(* IEC 61131-3 sources: ics/BLR101_ProenixContact/BLR101_1_ILC171_44/LogicalPOUs/Valve, 2 files *)

(* ---- ValveFB.ST ---- *)
(*@PROPERTIES_EX@
TYPE: POU
LOCALE: 0
IEC_LANGUAGE: ST
PLC_TYPE: independent
PROC_TYPE: independent
GROUP: Valve
*)
(*@KEY@:DESCRIPTION*)

(*@KEY@:END_DESCRIPTION*)
FUNCTION_BLOCK ValveFB

(*Group:Default*)

VAR
    Fb_Alrm_Tmr :	TON;
END_VAR

VAR_IN_OUT
    Vlv_strct :	Vlv;
END_VAR

VAR
    AlrmNotMove :	BOOL;
    AlrmSQ :	BOOL;
    RunManual :	BOOL;
    RunAuto :	BOOL;
    COM_Open :	BOOL;
    COM_Close :	BOOL;
END_VAR

VAR_INPUT
    SetOvertime :	TIME;
    Cycle :	Cycle;
END_VAR

VAR
    NotMove_Alrm_Tmr :	TON;
    AlrmFeedBack :	BOOL;
    AlarmBlock :	BOOL;
END_VAR

(*@KEY@: WORKSHEET
NAME: ValveFB
IEC_LANGUAGE: ST
*)
    (*Alarm processing*)
Fb_Alrm_Tmr(IN:=Vlv_strct.CW.Enable and (COM_Close or COM_Open) and not
    Vlv_strct.SW.RUN, PT:=t#3s);

NotMove_Alrm_Tmr(IN:=Vlv_strct.CW.Enable and
    ((COM_Close and not Vlv_strct.SW.Closed) or
    (COM_Open and not Vlv_strct.SW.Opened)),PT:=SetOvertime);

if Fb_Alrm_Tmr.Q then
    AlrmFeedBack:=true;
end_if;

if NotMove_Alrm_Tmr.Q then
    AlrmNotMove:=true;
end_if;

if (not Vlv_strct.CW.ExtraEn and (Vlv_strct.SW.COM_Open or Vlv_strct.SW.COM_Close)) then
    AlarmBlock:= true;
end_if;

if Vlv_strct.SW.Opened and Vlv_strct.SW.Closed then
    AlrmSQ:=true;
end_if;

if AlrmNotMove or AlrmSQ or AlrmFeedBack or Vlv_strct.CW.ExtraAlarm then
    Vlv_strct.SW.AlarmAccum:=true;
end_if;

if Vlv_strct.CW.ACK then
    Vlv_strct.SW.AlarmAccum:=false;
    AlrmFeedBack:=false;
    AlrmSQ:=false;
    AlrmnotMove:=false;
    AlarmBlock:= false;
end_if;

    (*Auto/Manual mode selection*)
if Vlv_strct.CW.EnableAuto then
    Vlv_strct.SW.Auto:= true;
end_if;
if Vlv_strct.CW.DisableAuto then
    Vlv_strct.SW.Auto:= false;
end_if;

Vlv_strct.SW.ManOK:=not Vlv_strct.SW.AlarmAccum and Vlv_strct.CW.AuxON and
    Vlv_strct.CW.Enable and not Vlv_strct.SW.Auto;

Vlv_strct.SW.AutoOK:= not Vlv_strct.SW.AlarmAccum and Vlv_strct.CW.AuxON and
    Vlv_strct.CW.Enable and Vlv_strct.SW.Auto and Cycle.SW.Running;

    (*Manual mode activation*)
if Vlv_strct.CW.ManOpen or Vlv_strct.CW.ManClose then
    RunManual:=true;
end_if;

if Vlv_strct.CW.Stop or not Vlv_strct.SW.ManOK then
    RunManual:=false;
end_if;

    (*Auto mode activation*)
RunAuto:= (Cycle.CW.PulseStart or RunAuto) and Vlv_strct.SW.AutoOK and
    Vlv_strct.SW.Auto;

    (*Set command for start*)
COM_Open:=((Vlv_strct.CW.AutoOpen and RunAuto and Vlv_strct.SW.AutoOK) or
    ((Vlv_strct.CW.ManOpen or COM_Open) and RunManual and Vlv_strct.SW.ManOK)) and not
    COM_Close and not Vlv_strct.SW.Opened;

COM_Close:=((Vlv_strct.CW.AutoClose and RunAuto and Vlv_strct.SW.AutoOK) or
    ((Vlv_strct.CW.ManClose or COM_Close) and RunManual and Vlv_strct.SW.ManOK)) and not
    COM_Open and not Vlv_strct.SW.Closed;

Vlv_strct.SW.COM_Open:=COM_Open and not Vlv_strct.CW.SimEn;
Vlv_strct.SW.COM_Close:=COM_Close and not Vlv_strct.CW.SimEn;

    (*Status processing*)
if Vlv_strct.SW.AlarmAccum then
    Vlv_strct.Status:=word#4;
elsif not Vlv_strct.CW.ExtraEn then
    Vlv_strct.Status:=word#8;
elsif Vlv_strct.SW.Opened then
    Vlv_strct.Status:=word#1;
elsif Vlv_strct.SW.Closed then
    Vlv_strct.Status:=word#2;
else
    Vlv_strct.Status:=word#0;
end_if;

Vlv_strct.CW.EnableAuto:=false;
Vlv_strct.CW.DisableAuto:=false;
Vlv_strct.CW.ManOpen:=false;
Vlv_strct.CW.Stop:=false;
Vlv_strct.CW.ManClose:=false;
Vlv_strct.CW.ACK:=false;

(*@KEY@: END_WORKSHEET *)
END_FUNCTION_BLOCK

(* ---- Valve_section.ST ---- *)
(*@PROPERTIES_EX@
TYPE: POU
LOCALE: 0
IEC_LANGUAGE: ST
PLC_TYPE: independent
PROC_TYPE: independent
GROUP: Valve
*)
(*@KEY@:DESCRIPTION*)

(*@KEY@:END_DESCRIPTION*)
PROGRAM Valve_section

(*Group:Default*)

VAR
    Vlv_Blr_in :	ValveFB;
    Vlv_Blr_out :	ValveFB;
    Exhsr_Gate :	ValveFB;
END_VAR

VAR_EXTERNAL
    Boiler :	Blr;
    Cycle :	Cycle;
    xVlv_in_QM_ON :	BOOL;
    xVlv_in_Remote :	BOOL;
    xVlv_in_RUN :	BOOL;
    xVlv_in_TorqueSwAlrm :	BOOL;
    xVlv_in_Closed :	BOOL;
    xVlv_in_Opened :	BOOL;
    xVlv_out_QM_ON :	BOOL;
    xVlv_out_Remote :	BOOL;
    xVlv_out_RUN :	BOOL;
    xVlv_out_TorqueSwAlrm :	BOOL;
    xVlv_out_Closed :	BOOL;
    xVlv_out_Opened :	BOOL;
    xExhsrGt_QM_ON :	BOOL;
    xExhsrGt_Remote :	BOOL;
    xExhsrGt_RUN :	BOOL;
    xExhsrGt_Closed :	BOOL;
    xExhsrGt_Opened :	BOOL;
    xVlv_in_COM_OP :	BOOL;
    xVlv_in_COM_CL :	BOOL;
    xVlv_out_COM_OP :	BOOL;
    xVlv_out_COM_CL :	BOOL;
    xExhsrGt_COM_OP :	BOOL;
    xExhsrGt_COM_CL :	BOOL;
    arrMB_Srv1Data :	MB2_TCP_ARR_W_0_7167;
    ExhsrGatePos :	Snsr;
END_VAR

VAR
    ExhsrGatePID :	BACL_PID3P_T1_V0_10;
END_VAR

(*@KEY@: WORKSHEET
NAME: Valve_section
IEC_LANGUAGE: ST
*)

    (*Boiler Input Valve DI*)
Boiler.V[1].CW.Enable:= xVlv_in_Remote;
Boiler.V[1].CW.AuxON:= Cycle.CW.AuxON;
Boiler.V[1].CW.ExtraEn:= xVlv_in_QM_ON;
Boiler.V[1].CW.ExtraAlarm:= not xVlv_in_TorqueSwAlrm;
Boiler.V[1].SW.Rem:= xVlv_in_Remote;
Boiler.V[1].SW.RUN:= xVlv_in_RUN;
Boiler.V[1].SW.Closed:= xVlv_in_Closed;
Boiler.V[1].SW.Opened:= xVlv_in_Opened;

    (*Boiler Input Valve FB call*)
Vlv_Blr_in(Vlv_strct:=Boiler.V[1],SetOvertime:=t#80s,Cycle:=Cycle);
Boiler.V[1]:=Vlv_Blr_in.Vlv_strct;
    (*ModBusArray ControlWord Reset*)
arrMB_Srv1Data[1492]:=word#0;

    (*Boiler Input Valve D0*)
xVlv_in_COM_OP:= Boiler.V[1].SW.COM_Open;
xVlv_in_COM_CL:= Boiler.V[1].SW.COM_Close;

    (*Boiler Output Valve DI*)
Boiler.V[2].CW.Enable:= xVlv_out_Remote;
Boiler.V[2].CW.AuxON:= Cycle.CW.AuxON;
Boiler.V[2].CW.ExtraEn:= xVlv_out_QM_ON;
Boiler.V[2].CW.ExtraAlarm:= not xVlv_out_TorqueSwAlrm;
Boiler.V[2].SW.Rem:= xVlv_out_Remote;
Boiler.V[2].SW.RUN:= xVlv_out_RUN;
Boiler.V[2].SW.Closed:= xVlv_out_Closed;
Boiler.V[2].SW.Opened:= xVlv_out_Opened;

    (*Boiler Output Valve FB call*)
Vlv_Blr_out(Vlv_strct:=Boiler.V[2],SetOvertime:=t#80s,Cycle:=Cycle);
Boiler.V[2]:=Vlv_Blr_out.Vlv_strct;
    (*ModBusArray ControlWord Reset*)
arrMB_Srv1Data[1508]:=word#0;

    (*Boiler Output Valve D0*)
xVlv_out_COM_OP:= Boiler.V[2].SW.COM_Open;
xVlv_out_COM_CL:= Boiler.V[2].SW.COM_Close;

    (*Exhauser Gate DI*)
Boiler.V[3].CW.Enable:= xExhsrGt_Remote;
Boiler.V[3].CW.AuxON:= Cycle.CW.AuxON;
Boiler.V[3].CW.ExtraEn:= xExhsrGt_QM_ON;
Boiler.V[3].SW.Rem:= xExhsrGt_Remote;
Boiler.V[3].SW.RUN:= xExhsrGt_RUN;
Boiler.V[3].SW.Closed:= xExhsrGt_Closed;
Boiler.V[3].SW.Opened:= xExhsrGt_Opened;

    (*Exhauser Gate FB call*)
Exhsr_Gate(Vlv_strct:=Boiler.V[3],SetOvertime:=t#60s,Cycle:=Cycle);
Boiler.V[3]:=Exhsr_Gate.Vlv_strct;
    (*ModBusArray ControlWord Reset*)
arrMB_Srv1Data[1524]:=word#0;

    (*Exhsr Gate Valve D0*)
xExhsrGt_COM_OP:= Boiler.V[3].SW.COM_Open;
xExhsrGt_COM_CL:= Boiler.V[3].SW.COM_Close;

Boiler.V[3].ActPos:=ExhsrGatePos.RealValue;

    (*Exhsr Gate Valve PID*)
ExhsrGatePID(IN_xActivate:=Boiler.Reg[0].CW.En,
    IN_tCycleTime:=t#3s,
    IN_rSetPoint:=Boiler.Reg[0].SP,
    IN_rActValue:=Boiler.AI[15].RealValue,
    IN_rDeadBand:=Boiler.Reg[2].DeadBand,
    IN_rKR:=Boiler.Reg[0].Kp,
    IN_rTN:=Boiler.Reg[0].Tn,
    IN_rTV:=Boiler.Reg[0].Tv,
    IN_tRunningTime:=t#5s);

Boiler.V[3].CW.AutoOpen:=ExhsrGatePID.OUT_xUp;
Boiler.V[3].CW.AutoClose:=ExhsrGatePID.OUT_xDown;

(*@KEY@: END_WORKSHEET *)
END_PROGRAM
